Staubli VAL3: master.pjx

Parameters version=s7.8 stackSize=5000 millimeterUnit=true
Program file=start.pgx
Program file=stop.pgx
Data file=master.dtx
